# B&R Automation Studio project 305841_E00002_AM_0 (part 16)

#### LocalFunctions.st
```iecst
// Calculate the master and slave angles given cut parameters
FUNCTION_BLOCK fbPopulateCamTable
  // **** Condition inputs
  _numPasses := MAX(1, numPasses); // 1 or greater. Otherwise treat as 1
  _finalDepth := ABS(finalDepth); // must be positive
  _finishPassDepth := MIN(MAX(0.0, finishPassDepth), _finalDepth); // must be >= 0.0, <= final depth.
  _cutInAngle := ABS(cutInAngle); // must be positive
  _overCutAngle := ABS(overCutAngle); // must be positive

  // **** First entry in table is 0,0
  // Axes start at 0,0 (0 offset) at the same velocity (which will normally be zero)
  // Specify absolute positions
  camTable.Section[0].Mode := mcCAMSECTREF_ABSOLUTE;
  camTable.Section[0].MasterPoint := 0.0;
  camTable.Section[0].SlavePoint := 0.0;
  // slave to be at a constant velocity
  camTable.Section[0].FirstDerivative := 1.0; // velocity ratio
  camTable.Section[0].SecondDerivative := 0.0; // accel ratio
  // next point will be offset. Use polynomial for this -- good general case solution
  camTable.Section[0].Type := mcCAMSECTLAW_5TH_ORDER_POLYNOM;
  camTable.Section[0].InflectionPoint := 0.0; // not used for polynomial

  // **** Figure out pass depths and then resulting angles
  // Make cam table entries
  incrCutDepth := (_finalDepth - _finishPassDepth) / _numPasses;

  IF incrCutDepth > 0.0 THEN
    // normal case where finishing pass < final depth
    FOR passCount := 1 TO _numPasses DO
      // depth for this pass
      totalPassDepth := incrCutDepth * passCount;
      // Look up angle for the needed depth
      fbLookupAngle(xVal := totalPassDepth,
                     t1 := ADR(depthToAngle_T1),
                     t2 := ADR(depthToAngle_T2),
                     t3 := ADR(depthToAngle_T3));
      passAngle := fbLookupAngle.yVal;

      // At this point, we have the angle for this pass.
      // This angle is actually the offset angle between the axes.
      // The offset in practice should be negative, meaning the slave lags
      // behind the master by the amount of the offset.
      // Make an entry in the cam table
      // Each pass has an enrty to establish the pass depth,
      // and a second pass to make the cut, which is 1 revolution from the point the
      // depth is established, plus the overcut distance.
      // For a given pass, the first index/position is: ((pass number - 1) * 2) + 1
      // the second index/position is: first index + 1
      // For a given pass, the first master position is: (cutInAngle + pass number) + ((rev + overcut) * (pass number - 1))
      // the second master position is: first position + rev + overcut
      idx := ((passCount - 1) * 2) + 1; // zero based array index position

      // Establish an offset from previous position
      camTable.Section[idx].Mode := mcCAMSECTREF_ABSOLUTE;
      camTable.Section[idx].MasterPoint := (_cutInAngle * passCount) + ((360.0 + _overCutAngle) * (passCount - 1));
      camTable.Section[idx].SlavePoint := camTable.Section[idx].MasterPoint - passAngle;
      // slave to be at a constant velocity
      camTable.Section[idx].FirstDerivative := 1.0; // velocity ratio
      camTable.Section[idx].SecondDerivative := 0.0; // accel ratio
      // next point will be a stright section.
      camTable.Section[idx].Type := mcCAMSECTLAW_STRAIGHT_LINE;
      camTable.Section[idx].InflectionPoint := 0.0; // not used for straight line

      // Keep the offset for a revolution + the overcut distance
      camTable.Section[idx + 1].Mode := mcCAMSECTREF_ABSOLUTE;
      camTable.Section[idx + 1].MasterPoint := camTable.Section[idx].MasterPoint + (360.0 + _overCutAngle);
      camTable.Section[idx + 1].SlavePoint := camTable.Section[idx + 1].MasterPoint - passAngle;
      // slave to be at a constant velocity
      camTable.Section[idx + 1].FirstDerivative := 1.0; // velocity ratio
      camTable.Section[idx + 1].SecondDerivative := 0.0; // accel ratio
      // next point will establish a new offset, so use a polynomial
      camTable.Section[idx + 1].Type := mcCAMSECTLAW_5TH_ORDER_POLYNOM;
      camTable.Section[idx + 1].InflectionPoint := 0.0; // not used for polynomial
    END_FOR;
  ELSE
    // Special case where finishing pass was entered to be >= final depth.
    // Nothing to do, and this else is here for documentation and as
    // a place holder in case something ends up being needed.
    // The finishing pass is handled next, and will cover this case
    ;
  END_IF

  // **** Figure out finishing pass situation

  // If there is a finishing pass, then create cam entries for it

  // After the for loop, passCount will be 1 more than the number of passes.
  // Perfect for the finishing pass, or the retract entry.
  idx := ((passCount - 1) * 2) + 1; // zero based array index position
  IF _finishPassDepth > 0.0 THEN
    // There is a finishing pass
    // By definition, the finishing pass gets us to our final depth,
    // so regardless of the earlier passes, the finishing pass is always
    // at the offset to give the final depth.
    // Look up angle for the needed depth
    fbLookupAngle(xVal := _finalDepth,
                   t1 := ADR(depthToAngle_T1),
                   t2 := ADR(depthToAngle_T2),
                   t3 := ADR(depthToAngle_T3));
    passAngle := fbLookupAngle.yVal;

    // Establish an offset from previous position
    camTable.Section[idx].Mode := mcCAMSECTREF_ABSOLUTE;
    camTable.Section[idx].MasterPoint := (_cutInAngle * passCount) + ((360.0 + _overCutAngle) * (passCount - 1));
    camTable.Section[idx].SlavePoint := camTable.Section[idx].MasterPoint - passAngle;
    // slave to be at a constant velocity
    camTable.Section[idx].FirstDerivative := 1.0; // velocity ratio
    camTable.Section[idx].SecondDerivative := 0.0; // accel ratio
    // next point will be a stright section.
    camTable.Section[idx].Type := mcCAMSECTLAW_STRAIGHT_LINE;
    camTable.Section[idx].InflectionPoint := 0.0; // not used for straight line

    // Keep the offset for a revolution + the overcut distance
    camTable.Section[idx + 1].Mode := mcCAMSECTREF_ABSOLUTE;
    camTable.Section[idx + 1].MasterPoint := camTable.Section[idx].MasterPoint + (360.0 + _overCutAngle);
    camTable.Section[idx + 1].SlavePoint := camTable.Section[idx + 1].MasterPoint - passAngle;
    // slave to be at a constant velocity
    camTable.Section[idx + 1].FirstDerivative := 1.0; // velocity ratio
    camTable.Section[idx + 1].SecondDerivative := 0.0; // accel ratio
    // next point will establish a new offset, so use a polynomial
    camTable.Section[idx + 1].Type := mcCAMSECTLAW_5TH_ORDER_POLYNOM;
    camTable.Section[idx + 1].InflectionPoint := 0.0; // not used for polynomial

    // increment the pass count so similar it can be used for the last entry
    passCount := passCount + 1;
    // calculate a new index for the last entry, which retracts the cutter
    idx := ((passCount - 1) * 2) + 1; // zero based array index position
  END_IF;

  // **** Do the last entry to retract the cutting head.
  // passCount will either be number of passes + 1 in the non-finishing pass case,
  // or will be number of passes + 2 in the finishing pass case. idx and passCount
  // were already adjusted in the finishing pass case.

  // The last cam entry needs to be of type mcCAMSECTLAW_LAST_POINT
  // Establish a zero offset from previous position
  camTable.Section[idx].Mode := mcCAMSECTREF_ABSOLUTE;
  camTable.Section[idx].MasterPoint := (_cutInAngle * passCount) + ((360.0 + _overCutAngle) * (passCount - 1));
  camTable.Section[idx].SlavePoint := camTable.Section[idx].MasterPoint;
  // slave to be at a constant velocity
  camTable.Section[idx].FirstDerivative := 1.0; // velocity ratio
  camTable.Section[idx].SecondDerivative := 0.0; // accel ratio
  // next point will be a stright section.
  camTable.Section[idx].Type := mcCAMSECTLAW_LAST_POINT;
  camTable.Section[idx].InflectionPoint := 0.0; // not used for straight line

END_FUNCTION_BLOCK

FUNCTION_BLOCK fbLookUpYValT3
  // See what table the x value is in
  tableNumber := fctGetTableNumberT3(xVal, ADR(t1), ADR(t2), ADR(t2));
  // Look up the angle (y value) from the correct table
  // The fbDepthToAngle will interpolate between table entries
  IF 1 = tableNumber THEN
    // Set up the lookup fb
    fbDepthToAngleLu(Enable := FALSE);
    fbDepthToAngleLu.NumberOfNodes := t1.numberOfVals;
    fbDepthToAngleLu.NodeVectorX := t1.xVals;
    fbDepthToAngleLu.FcnValues := t1.yVals;
    fbDepthToAngleLu.InX := xVal;
    // look up the Y value
    fbDepthToAngleLu(Enable := TRUE);
    IF fbDepthToAngleLu.Enable AND NOT fbDepthToAngleLu.Error THEN
      // Lookup worked. Send out the looked up value.
      yVal := fbDepthToAngleLu.Out;
    ELSE
      // Lookup didn't work. Send ou the sentinel value.
      yVal := INVALID_SENTINEL;
    END_IF;

  ELSIF 2 = tableNumber THEN
    // Set up the lookup fb
    fbDepthToAngleLu(Enable := FALSE);
    fbDepthToAngleLu.NumberOfNodes := t2.numberOfVals;
    fbDepthToAngleLu.NodeVectorX := t2.xVals;
    fbDepthToAngleLu.FcnValues := t2.yVals;
    fbDepthToAngleLu.InX := xVal;
    // look up the Y value
    fbDepthToAngleLu(Enable := TRUE);
    IF fbDepthToAngleLu.Enable AND NOT fbDepthToAngleLu.Error THEN
      // Lookup worked. Send out the looked up value.
      yVal := fbDepthToAngleLu.Out;
    ELSE
      // Lookup didn't work. Send ou the sentinel value.
      yVal := INVALID_SENTINEL;
    END_IF;

  ELSIF 3 = tableNumber THEN
    // Set up the lookup fb
    fbDepthToAngleLu(Enable := FALSE);
    fbDepthToAngleLu.NumberOfNodes := t3.numberOfVals;
    fbDepthToAngleLu.NodeVectorX := t3.xVals;
    fbDepthToAngleLu.FcnValues := t3.yVals;
    fbDepthToAngleLu.InX := xVal;
    // look up the Y value
    fbDepthToAngleLu(Enable := TRUE);
    IF fbDepthToAngleLu.Enable AND NOT fbDepthToAngleLu.Error THEN
      // Lookup worked. Send out the looked up value.
      yVal := fbDepthToAngleLu.Out;
    ELSE
      // Lookup didn't work. Send ou the sentinel value.
      yVal := INVALID_SENTINEL;
    END_IF;
  END_IF;

END_FUNCTION_BLOCK

// Given an X, find which of 3 tables to look in
FUNCTION fctGetTableNumberT3
  // Return a 1, 2, or 3 for which table to look in
  // NOTE: X values in each table need to be sorted in ascending order
  // NOTE: It is assumed that x values in table 1 < table 2 < table 3

  // If value is less than or equal the last value in table 1,
  // then the value must represented in or before table 1. Return 1.
  IF xVal <= t1.xVals[t1.numberOfVals - 1] THEN
    fctGetTableNumberT3 := 1;
    RETURN;
  ELSIF xVal >= t3.xVals[0] THEN
    // If value is greater than or equal to the first value in table 3,
    // then the value must be represented in or after table 3. Return 3.
    fctGetTableNumberT3 := 3;
    RETURN;
  ELSE
    // The value must be too big to be represented in table 1,
    // and too small to be represented in table 3.
    // Table 2 is the best choice. Return 2.
    fctGetTableNumberT3 := 2;
    RETURN;
  END_IF;

END_FUNCTION

// Given a table, swap the X and Y values
FUNCTION fctSwapTableT3
  // Make sure number of values does not overrun the array sizes
  length := MIN(SIZEOF(tVals) / SIZEOF(tVals[0]), SIZEOF(table.xVals) / SIZEOF(table.xVals[0]), SIZEOF(table.yVals) / SIZEOF(table.yVals[0]));
  // Y -> temp
  // X -> Y
  // temp -> X
  // nextAddr := brsmemcpy(ADR(Dest),ADR(Src),length);
  nextAddr := brsmemcpy(ADR(tVals), ADR(table.yVals), length);
  nextAddr := brsmemcpy(ADR(table.yVals), ADR(table.xVals), length);
  nextAddr := brsmemcpy(ADR(table.xVals), ADR(tVals), length);
END_FUNCTION
```

### Library Logical/PlcLogic/CutProfile/CreateCamTable

#### CreateCamTable.var
```iecst
VAR CONSTANT
  CAM_POINTS : UINT := 250;
END_VAR

VAR

  (* program control *)
  seqCtr : SINT; (* sequence counter *)
  idx : UINT; (* index *)

  (****** Cam related ******)
  (* program control for cam creation *)
  reqCreateCamTable : BOOL := FALSE; (* request to start seq *)
  createCamTableOS : BOOL := FALSE;
  createCamTableDone : BOOL := FALSE;
  camTableId : UINT := 14; (* 1-14, but data type compatible with cam prepare fb *)
  camSeqCtr : SINT; (* sequence counter *)
  camTable : McCamSectionsType; (* local cam sections table *)
  camData : McCamDataType; (* cam data calculated from sections *)
  camPointsMaster : ARRAY[0..CAM_POINTS] OF LREAL;
  camPointsSlave : ARRAY[0..CAM_POINTS] OF LREAL;
  fbCreateCamSections : fbCalcCamSections;
  fbCalcCamFromSections : MC_BR_CalcCamFromSections;
  fbCalcCamPoints : MC_BR_CalcPointsFromCam;
  fbCamPrepare : MC_BR_CamPrepare;
  (* detect changes to cut profile *)
  cutProfilePrev : sWp_CuttingHead;
  (* BR Str mem fct params *)
  cutProfileBytes : UDINT;
  result : DINT;
  nxtAddr : UDINT;

  (****** Recipe and file related ******)

  (* Local version OF the lookup table *)
	depthToAngleLu : sDepthToAngleLu;

  (* program control for directory creation *)
  reqInitDirs : BOOL := FALSE; (* request to start seq *)
  initDirsOS : BOOL := FALSE;
  initDirsDone : BOOL := FALSE;
  devName : STRING[80]; (* also used for recipe read *)
  dirName : STRING[255];

  (* program control for Depth To Angle Lu recipe registration *)
  pvNameLocalDepthToAngleLu : STRING[100];
  pvNameGloballDepthToAngleLu : STRING[100];
  pvCatagoryDepthToAngleLu : STRING[50];

  (* program control for recipe read/write *)
  recipeReadOverwiteGlobal : BOOL := FALSE;

  recipeReadFileName : STRING[255];
  recipeWriteFileName : STRING[255];

  reqRecipeReadAngleLu : BOOL := FALSE;
  recipeReadAngleLuOS : BOOL := FALSE;
  recipeReadAngleLuDone : BOOL := FALSE;

  reqRecipeWriteAngleLu : BOOL := FALSE;
  recipeWriteAngleLuOS : BOOL := FALSE;
  recipeWriteAngleLuDone : BOOL := FALSE;
  csvHeader : MpRecipeCsvHeaderType;

  (* FileIO fbs *)
  fbDirCreate : DirCreate;

  (* recipe fbs *)
  fbRcpiRegLocalDToALu : MpRecipeRegPar; (* register local Depth To Angle Lu Table to recipe *)
  fbRcpiRegGlobalDToALu : MpRecipeRegPar; (* register global Depth To Angle Lu Table to recipe *)
  fbRecipeCsv : MpRecipeCsv; (* recipe to/from file *)

END_VAR
```

#### LocalFunctions.fun
```iecst
FUNCTION_BLOCK fbLookUpYValT3 (* Given an X, get the possibly interpolated value for Y *)
	VAR CONSTANT
		INVALID_SENTINEL : REAL := -9999.0;
	END_VAR

	VAR_INPUT
    LoadTables : BOOL; (* load lookup table values *)
    Enable : BOOL; (* trigger a lookup *)
		XVal : REAL; (* x value to lookup *)
		T1 : REFERENCE TO sXYTableReal50; (* table 1 *)
		T2 : REFERENCE TO sXYTableReal50; (* table 2 *)
		T3 : REFERENCE TO sXYTableReal50; (* table 3 *)
	END_VAR

	VAR_OUTPUT
    IsTablesLoaded : BOOL; (* look up tables have been loaded *)
    Active : BOOL;
    Done : BOOL;
    Error : BOOL;
		YVal : REAL; (* looked up and interpolated Y value *)
	END_VAR

	VAR
    (* oneshots *)
    _loadOS : BOOL := FALSE;
    _enableOS : BOOL := FALSE;
    (* which table to use *)
		_xValPrev : REAL; (* previous x value to lookup *)
    _tableNumber : USINT;
    (* table lookup fbs*)
		_fbDepthToAngleLuT1 : MTLookUpTable;
		_fbDepthToAngleLuT2 : MTLookUpTable;
		_fbDepthToAngleLuT3 : MTLookUpTable;
	END_VAR
END_FUNCTION_BLOCK

FUNCTION_BLOCK fbPopulateCamSections (* Calculate the master and slave angles given cut parameters *)
	VAR_INPUT
    Enable : BOOL;
		PassCount : USINT := 1; (* number of passes *)
		FinalDepth : REAL; (* final cut depth, in units of lookup table *)
		FinishPassDepth : REAL := 0.0; (* finishing pass depth. In units of lookup table. Set to 0 for no finish pass. *)
		CutInAngle : REAL; (* degrees *)
		OverCutAngle : REAL; (* degrees *)
		CamTable : REFERENCE TO McCamSectionsType; (* X values master angle, Y values slave angle *)
		DepthToAngle_T1 : REFERENCE TO sXYTableReal50;
		DepthToAngle_T2 : REFERENCE TO sXYTableReal50;
		DepthToAngle_T3 : REFERENCE TO sXYTableReal50;
	END_VAR

  VAR_OUTPUT
    Active : BOOL := FALSE;
    Done : BOOL := FALSE;
    Error : BOOL := FALSE;
  END_VAR

	VAR
    enableOS : BOOL := FALSE;
		_numPasses : USINT; (* conditioned number of passes *)
		_finalDepth : REAL; (* conditioned final cut depth *)
		_finishPassDepth : REAL; (* conditioned finishing pass depth. Set to 0 for no finish pass. *)
		_cutInAngle : REAL; (* conditioned value *)
		_overCutAngle : REAL; (* conditioned value *)
    seqCtr : SINT; (* sequence counter *)
		passCtr : USINT; (* pass counter *)
		incrCutDepth : REAL; (* incremental depth of a nominal pass *)
		totalPassDepth : REAL; (* accum depth for the pass *)
		passAngle : REAL;
		idx : USINT; (* index *)
    (* lookup angle from depth fb *)
    fbLookupAngle : fbLookUpYValT3;
	END_VAR
END_FUNCTION_BLOCK

FUNCTION fctGetTableNumberT3 : USINT (* Given an X, find which table to look in *)
	VAR_INPUT
		xVal : REAL;
		t1 : REFERENCE TO sXYTableReal50; (* table 1 *)
		t2 : REFERENCE TO sXYTableReal50; (* table 2 *)
		t3 : REFERENCE TO sXYTableReal50; (* table 3 *)
	END_VAR
END_FUNCTION

FUNCTION fctSwapTableT3 : USINT (* Swap X & Y columns *)
	VAR_INPUT
		table : REFERENCE TO sXYTableReal50; (* table to swap the X & Y values of *)
	END_VAR
	VAR
		tVals : ARRAY[0..49] OF REAL; (* temporary storage *)
		length : UDINT; (* mem copy length in bytes *)
		nextAddr : UDINT; (* return from memcpy *)
	END_VAR
END_FUNCTION
```

#### CreateCamTable.st
```iecst
PROGRAM _INIT

  (****** Cam related ******)
  // Set up fb to populate cam sections
  fbCreateCamSections.CamTable := ADR(camTable);
  fbCreateCamSections.DepthToAngle_T1 := ADR(gr_depthToAngleLu.T1);
  fbCreateCamSections.DepthToAngle_T2 := ADR(gr_depthToAngleLu.T2);
  fbCreateCamSections.DepthToAngle_T3 := ADR(gr_depthToAngleLu.T3);

  (****** Recipe and file related ******)
  gr_depthToAngleLu; // Make sure the tables exist!!
  depthToAngleLu;

  // Setup registration of PV to a recipe
  // Each PV uses a separate registration FB
  // Local Depth To Angle LU Table
  // Use local LU table for recipe access and transfer to/from global when all is well
  pvNameLocalDepthToAngleLu := 'CrCamTbl:depthToAngleLu';
  pvCatagoryDepthToAngleLu := 'DepthToAngle';
  fbRcpiRegLocalDToALu.MpLink := ADR(angleLuRecipeCsv);
  fbRcpiRegLocalDToALu.Enable := FALSE;
  fbRcpiRegLocalDToALu.ErrorReset := FALSE;
  fbRcpiRegLocalDToALu.PVName := ADR(pvNameLocalDepthToAngleLu);
  fbRcpiRegLocalDToALu.Category := ADR(pvCatagoryDepthToAngleLu);
  // set up the fb by calling with enable false, and then set enable
  // true so it is ready to go in cyclic.
  fbRcpiRegLocalDToALu();
  fbRcpiRegLocalDToALu.Enable := TRUE;

  // Global Depth To Angle LU Table
  // Use local LU table for recipe access and transfer to/from global when all is well
  pvNameGloballDepthToAngleLu := 'gr_depthToAngleLu';
  pvCatagoryDepthToAngleLu := 'DepthToAngle';
  fbRcpiRegGlobalDToALu.MpLink := ADR(angleLuRecipeCsv);
  fbRcpiRegGlobalDToALu.Enable := FALSE;
  fbRcpiRegGlobalDToALu.ErrorReset := FALSE;
  fbRcpiRegGlobalDToALu.PVName := ADR(pvNameGloballDepthToAngleLu);
  fbRcpiRegGlobalDToALu.Category := ADR(pvCatagoryDepthToAngleLu);
  // set up the fb by calling with enable false, and then set enable
  // true so it is ready to go in cyclic.
  fbRcpiRegGlobalDToALu();
  fbRcpiRegGlobalDToALu.Enable := TRUE;

  // Set flag to create directories
  initDirs := TRUE; // true will trigger dir setup (creation) after startup
  initDirsOS := FALSE;
  initDirsDone := FALSE;

  // Set flags to control read/write of recipes
  // recipe file names
  recipeReadFileName := 'DepthToAngleLookup_recipe_b.csv';
  recipeWriteFileName := 'DepthToAngleLookup_recipe_b_FromPlc.csv';

  // set whether or not to overwrite the global data on sucessful local read
  recipeReadOverwiteGlobal := FALSE;

  recipeReadAngleLu := FALSE; // set high to read recipe after startup
  recipeReadAngleLuOS := FALSE;
  recipeReadAngleLuDone := FALSE;

  recipeWriteAngleLu := FALSE; // set high to read recipe after startup
  recipeWriteAngleLuOS := FALSE;
  recipeWriteAngleLuDone := FALSE;

 END_PROGRAM

PROGRAM _CYCLIC

  // *****************
  // Create Cam table on request
  // *****************

  // On request, calculate and populate cam sections base on cut parameters.
  // Done sucessfully, and camSeqCtr should start from 1, go up, and then end up at -1.
  // Errors result in a more negative camSeqCtr
  // TODO: Deal with errors. Right now the sequence stops, with the camSeqCtr being set to
  // a value more negative than -1.

  IF createCamTable THEN

    // if the OS is clear, this is the first time thru ...
    // init the seq number and manage flags and OS
    IF NOT createCamTableOS THEN
      // Set the OS so this bit only happens once per req
      createCamTableOS := TRUE;
      // Init the seq ctr
      camSeqCtr := 1;
      // Clear the done flag
      createCamTableDone := FALSE;
    END_IF;

    IF 1 = camSeqCtr THEN
      // Use cam id 14 for calculated cam table
      camTableId := 14;

      // Set up to calc the cam sections fb
      // Use the current cutting head configuration for the cut profile

      // Force the finish pass depth to be zero if the option is not chosen
      IF gr_CfgCurrent.cuttingHead.finishingPass THEN
        fbCreateCamSections.FinishPassDepth :=  gr_CfgCurrent.cuttingHead.finishingPassDepth;
      ELSE
        fbCreateCamSections.FinishPassDepth := 0.0;
      END_IF;
      fbCreateCamSections.PassCount := gr_CfgCurrent.cuttingHead.passCount;
      fbCreateCamSections.FinalDepth := gr_CfgCurrent.cuttingHead.totalDepth;
      fbCreateCamSections.CutInAngle :=  LREAL_TO_REAL(gr_CfgCurrent.cuttingHead.depthAdjAngle);
      fbCreateCamSections.OverCutAngle :=  LREAL_TO_REAL(gr_CfgCurrent.cuttingHead.cutOverrunAngle);

      // Clear the camTable, camData, and point arrays
      // nxt_adr := brsmemset(ADR(Mem),value,length);
      nxtAddr := brsmemset(ADR(camTable), 0, SIZEOF(camTable));
      nxtAddr := brsmemset(ADR(camData), 0, SIZEOF(camData));
      nxtAddr := brsmemset(ADR(camPointsMaster), 0, SIZEOF(camPointsMaster));
      nxtAddr := brsmemset(ADR(camPointsSlave), 0, SIZEOF(camPointsSlave));

      // Call with enable false to make sure everything is reset and ready to execute with new info
      fbCreateCamSections.Enable := FALSE;
      fbCreateCamSections();
      // onto the next step
      camSeqCtr := 2;
    ELSIF 2 = camSeqCtr THEN
      // Calc the cam sections
      fbCreateCamSections.Enable := TRUE;
      fbCreateCamSections();
      IF fbCreateCamSections.Done AND NOT fbCreateCamSections.Error THEN
        // All done and no error. Move on ...
        // Reset FB and go to next step
        fbCreateCamSections.Enable := FALSE;
        fbCreateCamSections();
        camSeqCtr := 3;
      ELSIF fbCreateCamSections.Done AND fbCreateCamSections.Error THEN
        // Done with an error. Bail out ...
        camSeqCtr := -2;
      END_IF;
    ELSIF 3 = camSeqCtr THEN
      // Set up to calc the cam from the sections
      fbCalcCamFromSections.CamSectionsAddress := ADR(camTable);
      fbCalcCamFromSections.CamDataAddress := ADR(camData);
      // Call with execute false to make sure everything is reset and ready to execute with new info
      fbCalcCamFromSections.Execute := FALSE;
      fbCalcCamFromSections();
      // onto the next step
      camSeqCtr := 4;
    ELSIF 4 = camSeqCtr THEN
      // Calc the cam sections
      fbCalcCamFromSections.Execute := TRUE;
      fbCalcCamFromSections();
      IF fbCalcCamFromSections.Done AND NOT fbCalcCamFromSections.Error THEN
        // All done and no error. Move on ...
        // Reset FB and go to next step
        fbCalcCamFromSections.Execute := FALSE;
        fbCalcCamFromSections();
        camSeqCtr := 5;
      ELSIF NOT fbCalcCamFromSections.Busy AND fbCalcCamFromSections.Error THEN
        // Done with an error. Bail out ...
        camSeqCtr := -4;
      END_IF;
    ELSIF 5 = camSeqCtr THEN
      // Set up to prepare and load the cam data
      fbCamPrepare.Axis := ADR(axes[AD_INNER_ECCENTRIC].AxisObj);
      fbCamPrepare.Cam.DataObjectName := ''; // not used if Cam.DataAdress <> 0
      fbCamPrepare.Cam.DataAdress := ADR(camData); // cam data calculated in fbCalcCamFromSections
      fbCamPrepare.CamID := camTableId;
      // Call with execute false to make sure everything is reset and ready to execute with new info
      fbCamPrepare.Execute := FALSE;
      fbCamPrepare();
      // onto the next step
      camSeqCtr := 6;
    ELSIF 6 = camSeqCtr THEN
      // Prepare and load the cam data
      fbCamPrepare.Execute := TRUE;
      fbCamPrepare();
      IF fbCamPrepare.Done AND NOT fbCamPrepare.Error THEN
        // All done and no error. Move on ...
        // Reset FB and go to next step
        fbCamPrepare.Execute := FALSE;
        fbCamPrepare();
        camSeqCtr := -1;  // TEST: skip fbCalcCamPoints. Getting an error
      ELSIF NOT fbCamPrepare.Busy AND fbCamPrepare.Error THEN
        // Done with an error. Bail out ...
        camSeqCtr := -6;
      END_IF;
    ELSIF 7 = camSeqCtr THEN
      // Set up to calculate cam points
      fbCalcCamPoints.Cam.DataObjectName := ''; // not used if Cam.DataAdress <> 0
      fbCalcCamPoints.Cam.DataAdress := ADR(camData); // cam data calculated in fbCalcCamFromSections
      fbCalcCamPoints.MasterPointsAddress := ADR(camPointsMaster);
      fbCalcCamPoints.SlavePointsAddress := ADR(camPointsSlave);
      fbCalcCamPoints.NumberOfPoints := CAM_POINTS;
      // Call with execute false to make sure everything is reset and ready to execute with new info
      fbCalcCamPoints.Execute := FALSE;
      fbCalcCamPoints();
      // onto the next step
      camSeqCtr := 8;
    ELSIF 8 = camSeqCtr THEN
      // Calcuate points from the cam data
      fbCalcCamPoints.Execute := TRUE;
      fbCalcCamPoints();
      IF fbCalcCamPoints.Done AND NOT fbCalcCamPoints.Error THEN
        // All done and no error. Move on ...
        // reset fb
        fbCalcCamPoints.Execute := FALSE;
        fbCalcCamPoints();
        camSeqCtr := -1;
      ELSIF NOT fbCalcCamPoints.Busy AND fbCalcCamPoints.Error THEN
        // Done with an error. Bail out ...
        camSeqCtr := -8;
      END_IF;
    ELSIF -1 = camSeqCtr THEN
      // All done making cam sections.
      // Getting ready if another request is made.
      // Clear the createCamTable flag and OS and set the done.
     createCamTable := FALSE;
     createCamTableOS := FALSE; // clear the OS so another initDirs resets things up top
     createCamTableDone := TRUE;
     // reset fb
     fbCreateCamSections.Enable := FALSE;
     fbCreateCamSections();
    END_IF;
  ELSE
    // createCamTable is false. Clear the OS so we can one time thru it next time
    createCamTableOS := FALSE;
  END_IF;

  // *****************
  // Set up directories
  // *****************
  // Execute FileIO DirCreate async until done or error
  // seqCtr odd: set up DirCreate fb
  // seqCtr even : create dir
  // Use the OS so the directory management can be easily re-run
  // by setting initDirs true (again)
  IF initDirs THEN
    // if the OS is clear, this is the first time thru ...
    // init the seq number and manage flags and OS
    IF NOT initDirsOS THEN
      // Set the OS so this bit only happens once per initDirs
      initDirsOS := TRUE;
      // Init the seq ctr
      seqCtr := 1;
      // Clear the done flag
      initDirsDone := FALSE;
    END_IF;

    IF 1 = seqCtr THEN
      // Setup for first dir
      devName := 'UserPartitionRoot';
      dirName := 'config';
      fbDirCreate.enable := FALSE;
      fbDirCreate.pDevice := ADR(devName);
      fbDirCreate.pName := ADR(dirName);
      fbDirCreate();
      IF ERR_FUB_ENABLE_FALSE = fbDirCreate.status THEN
        seqCtr := 2;
      END_IF;
    ELSIF 2 = seqCtr THEN
      // create first dir
      fbDirCreate.enable := TRUE;
      fbDirCreate();
      IF ERR_OK = fbDirCreate.status OR fiERR_DIR_ALREADY_EXIST = fbDirCreate.status THEN
        // creation okay or not needed
        seqCtr := 3;
      END_IF;
    ELSIF 3 = seqCtr THEN
      // Setup for seconnd dir
      dirName := 'config\recipes';
      // same addresses for device and name
      fbDirCreate.enable := FALSE;
      fbDirCreate();
      IF ERR_FUB_ENABLE_FALSE = fbDirCreate.status THEN
        seqCtr := 4;
      END_IF;
    ELSIF 4 = seqCtr THEN
      // create second dir
      fbDirCreate.enable := TRUE;
      fbDirCreate();
      IF ERR_OK = fbDirCreate.status OR fiERR_DIR_ALREADY_EXIST = fbDirCreate.status THEN
        // creation okay or not needed
        seqCtr := -1;
      END_IF;
    ELSIF -1 = seqCtr THEN
      // All done making directories.
      // Getting ready if another request is made.
      // Clear the initDirs flag and OS and set the done.
     initDirs := FALSE;
     initDirsOS := FALSE; // clear the OS so another initDirs resets things up top
     initDirsDone := TRUE;
     // shut off the fb as a matter of good practice
     fbDirCreate.enable := FALSE;
     fbDirCreate();
    END_IF;
  ELSE
    // initDirs is false. Clear the OS so we can one time thru it next time
    initDirsOS := FALSE;
  END_IF;

  // *****************
  // Read Write Lu Tables to/from recipe
  // *****************

  // Recipe Registration fb should be called all the time, and need to be active
  // when recipe read/write is performed.
  // MpRecipeRegPar was set up in init
  fbRcpiRegLocalDToALu();
  fbRcpiRegGlobalDToALu();

  // **** Read Recipe
  // Treat recipe read as async until done or error
  // seqCtr odd: set up fbRecipeCsv fb
  // seqCtr even : read recipe
  // Use the OS so the read can be easily re-run
  // by setting registerPvs true (again)
  IF NOT initDirs AND initDirsDone AND
      fbRcpiRegLocalDToALu.Active AND NOT fbRcpiRegLocalDToALu.Error AND
      fbRcpiRegGlobalDToALu.Active AND NOT fbRcpiRegGlobalDToALu.Error AND
      recipeReadAngleLu AND NOT recipeWriteAngleLu THEN
    // if the OS is clear, this is the first time thru ...
    // init the seq number and manage flags and OS
    IF NOT recipeReadAngleLuOS THEN
      // Set the OS so this bit only happens once per initDirs
      recipeReadAngleLuOS := TRUE;
      // Set the pv number
      seqCtr := 1;
      // Clear the done flag
      recipeReadAngleLuDone := FALSE;
    END_IF;

    IF 1 = seqCtr THEN
      // Setup for first pv
      devName := 'Recipes';
      pvCatagoryDepthToAngleLu := 'DepthToAngle';
      fbRecipeCsv.MpLink := ADR(angleLuRecipeCsv);
      fbRecipeCsv.Enable := FALSE;
      fbRecipeCsv.ErrorReset := FALSE;
      fbRecipeCsv.DeviceName := ADR(devName);
      fbRecipeCsv.FileName := ADR(recipeReadFileName);
      fbRecipeCsv.Header := ADR(csvHeader);
      fbRecipeCsv.Category := ADR(pvCatagoryDepthToAngleLu);
      fbRecipeCsv.LoadType := mpRECIPE_CSV_LOAD_ALL;
      fbRecipeCsv.Load := TRUE;
      fbRecipeCsv.Save := FALSE;
      fbRecipeCsv.UpdateNotification := FALSE;
      fbRecipeCsv();
      IF NOT fbRecipeCsv.Enable AND NOT fbRecipeCsv.Active AND 0 = fbRecipeCsv.StatusID THEN
        seqCtr := 2;
      END_IF;
    ELSIF 2 = seqCtr THEN
      // read the recipe file and populate the pv
      fbRecipeCsv.Enable := TRUE;
      fbRecipeCsv();
      IF fbRecipeCsv.CommandDone AND NOT fbRecipeCsv.Error THEN
        // read ok
        // If the bit is set, transfer local to the global table -- thisglobal is battery backed retained/permanent
        IF recipeReadOverwiteGlobal THEN
          gr_depthToAngleLu := depthToAngleLu;
        END_IF;
        seqCtr := -1; // all done!
      END_IF;
    ELSIF -1 = seqCtr THEN
      // All done reading the recipe. Deal with flags
      recipeReadAngleLu := FALSE;
      recipeReadAngleLuOS := FALSE; // clear the OS so another registerPv resets things
      recipeReadAngleLuDone := TRUE;
      // shut off the fb as a matter of good practice
      fbRecipeCsv.Enable := FALSE;
      fbRecipeCsv();
    END_IF;
  ELSE
    // Earlier operations not done, or recipeReadAngleLu flag is clear. Clear to OS so we can one time thru it next time
    recipeReadAngleLuOS := FALSE;
  END_IF;

  // **** Write Recipe
  // Treat recipe read as async until done or error
  // seqCtr odd: set up fbRecipeCsv fb
  // seqCtr even : read recipe
  // Use the OS so the read can be easily re-run
  // by setting registerPvs true (again)
  IF NOT initDirs AND initDirsDone AND
      fbRcpiRegLocalDToALu.Active AND NOT fbRcpiRegLocalDToALu.Error AND
      fbRcpiRegGlobalDToALu.Active AND NOT fbRcpiRegGlobalDToALu.Error AND
      recipeWriteAngleLu AND NOT recipeReadAngleLu THEN
    // if the OS is clear, this is the first time thru ...
    // init the seq number and manage flags and OS
    IF NOT recipeWriteAngleLuOS THEN
      // Set the OS so this bit only happens once per initDirs
      recipeWriteAngleLuOS := TRUE;
      // Set the pv number
      seqCtr := 1;
      // Clear the done flag
      recipeWriteAngleLuDone := FALSE;
    END_IF;

    IF 1 = seqCtr THEN
      // Setup for first pv
      devName := 'Recipes';
      pvCatagoryDepthToAngleLu := 'DepthToAngle';
      csvHeader.Name := 'DepthToAngle';
      csvHeader.Description := 'Depths are given in inches, and angles correspond to negative (slave lag) offsets. Source is Robbie Potts Email.';
      csvHeader.Version := 'b';
      csvHeader.DateTime := DT#2022-06-03-14:56;
      fbRecipeCsv.MpLink := ADR(angleLuRecipeCsv);
      fbRecipeCsv.Enable := FALSE;
      fbRecipeCsv.ErrorReset := FALSE;
      fbRecipeCsv.DeviceName := ADR(devName);
      fbRecipeCsv.FileName := ADR(recipeWriteFileName);
      fbRecipeCsv.Header := ADR(csvHeader);
      fbRecipeCsv.Category := ADR(pvCatagoryDepthToAngleLu);
      fbRecipeCsv.LoadType := mpRECIPE_CSV_LOAD_ALL;
      fbRecipeCsv.Load := FALSE;
      fbRecipeCsv.Save := TRUE;
      fbRecipeCsv.UpdateNotification := FALSE;
      fbRecipeCsv();
      IF NOT fbRecipeCsv.Enable AND NOT fbRecipeCsv.Active AND 0 = fbRecipeCsv.StatusID THEN
        seqCtr := 2;
      END_IF;
    ELSIF 2 = seqCtr THEN
      // write pv to recipe file
      fbRecipeCsv.Enable := TRUE;
      fbRecipeCsv();
      IF fbRecipeCsv.CommandDone AND NOT fbRecipeCsv.Error THEN
        // read ok
        seqCtr := -1; // all done!
      END_IF;
    ELSIF -1 = seqCtr THEN
      // All done reading the recipe. Deal with flags
      recipeWriteAngleLu := FALSE;
      recipeWriteAngleLuOS := FALSE; // clear the OS so another registerPv resets things
      recipeWriteAngleLuDone := TRUE;
      // shut off the fb as a matter of good practice
      fbRecipeCsv.Enable := FALSE;
      fbRecipeCsv();
    END_IF;
  ELSE
    // Earlier operations not done, or recipeWriteAngleLu flag is clear. Clear to OS so we can one time thru it next time
    recipeWriteAngleLuOS := FALSE;
  END_IF;

END_PROGRAM

PROGRAM _EXIT
	(* Insert code here *)

END_PROGRAM
```

#### LocalFunctions.st
```iecst
FUNCTION_BLOCK fbLookUpYValT3
  // The lookup table needs to be loaded into the MTLookUpTable fb.
  // We don't want to do this every scan, so use the initTables to
  // trigger this, and the isInitialized output to monitor it.
  // Initialize the tables on a rising edge of initTables input,
  // OR if they have not been done yet and the enable goes high.

  IF (LoadTables AND NOT _loadOS) OR (Enable AND NOT IsTablesLoaded) THEN
    // Load tables if requested or if a lookup is triggered and they are not loaded.
    // First set the OS so only a rising edge of loadTables is used
    _loadOS := TRUE;
    // Now load the table values
    _fbDepthToAngleLuT1.NumberOfNodes := T1.numberOfVals;
    _fbDepthToAngleLuT1.NodeVectorX := T1.xVals;
    _fbDepthToAngleLuT1.FcnValues := T1.yVals;

    _fbDepthToAngleLuT2.NumberOfNodes := T2.numberOfVals;
    _fbDepthToAngleLuT2.NodeVectorX := T2.xVals;
    _fbDepthToAngleLuT2.FcnValues := T2.yVals;

    _fbDepthToAngleLuT3.NumberOfNodes := T3.numberOfVals;
    _fbDepthToAngleLuT3.NodeVectorX := T3.xVals;
    _fbDepthToAngleLuT3.FcnValues := T3.yVals;

    // set the output status
    IsTablesLoaded := TRUE;
  ELSIF NOT LoadTables THEN
    // keep OS false when init is not set
    _loadOS := FALSE;
  END_IF;

  // clear the done bit on rising edge of enable
  IF (Enable AND NOT _enableOS) OR (Enable AND XVal <> _xValPrev) THEN
    // first time thru with enable set, or enable is set and the x value changes

    // set the OS
    _enableOS := TRUE;

    // Clear the done bit and set the active bit
    Done := FALSE;
    Active := TRUE;

    // See what table the x value is in
    _tableNumber := fctGetTableNumberT3(XVal, ADR(T1), ADR(T2), ADR(T3));

    // Look up the Y value from the correct table
    // The fbDepthToAngle will interpolate between table entries
    // Call with correct lookup fb with enable false to make sure
    // input changes, including possible table updates above
    // are processed on rising edge of enable later on.
    IF 1 = _tableNumber THEN
      // Set up the lookup fb
      _fbDepthToAngleLuT1.InX := XVal;
      _fbDepthToAngleLuT1.Mode := mtLOOKUP_LINEAR_EXTRAPOLATION;
      _fbDepthToAngleLuT1(Enable := FALSE);
    ELSIF 2 = _tableNumber THEN
      // Set up the lookup fb
      _fbDepthToAngleLuT2.InX := XVal;
      _fbDepthToAngleLuT2.Mode := mtLOOKUP_LINEAR_EXTRAPOLATION;
      _fbDepthToAngleLuT2(Enable := FALSE);
    ELSIF 3 = _tableNumber THEN
      // Set up the lookup fb
      _fbDepthToAngleLuT3.InX := XVal;
      _fbDepthToAngleLuT3.Mode := mtLOOKUP_LINEAR_EXTRAPOLATION;
      _fbDepthToAngleLuT3(Enable := FALSE);
    END_IF;

    // Update the previos X value
    _xValPrev := XVal;

  ELSIF Enable AND _enableOS THEN
    // First time thru completed. Do this while enable is high.
    // LU FBs were set up on first scan thru, so now get on with
    // the lookup.
    IF 1 = _tableNumber THEN
      // look up the Y value from table 1
      _fbDepthToAngleLuT1(Enable := TRUE);
      IF _fbDepthToAngleLuT1.Enable AND _fbDepthToAngleLuT1.Active AND NOT _fbDepthToAngleLuT1.Error THEN
        // Lookup worked. Send out the looked up value.
        YVal := _fbDepthToAngleLuT1.Out;
        Error := FALSE;
      ELSIF _fbDepthToAngleLuT1.Enable AND _fbDepthToAngleLuT1.Error THEN
        // Lookup didn't work. Send out the sentinel value.
        YVal := INVALID_SENTINEL;
        Error := TRUE;
      END_IF;
      // All done, set the done output
      Done := TRUE;
    ELSIF 2 = _tableNumber THEN
      // look up the Y value from table 2
      _fbDepthToAngleLuT2(Enable := TRUE);
      IF _fbDepthToAngleLuT2.Enable AND _fbDepthToAngleLuT2.Active AND NOT _fbDepthToAngleLuT2.Error THEN
        // Lookup worked. Send out the looked up value.
        YVal := _fbDepthToAngleLuT2.Out;
        Error := FALSE;
      ELSIF _fbDepthToAngleLuT2.Enable AND _fbDepthToAngleLuT2.Error THEN
        // Lookup didn't work. Send out the sentinel value.
        YVal := INVALID_SENTINEL;
        Error := TRUE;
      END_IF;
      // All done, set the done output
      Done := TRUE;
    ELSIF 3 = _tableNumber THEN
      // look up the Y value from table 3
      _fbDepthToAngleLuT3(Enable := TRUE);
      IF _fbDepthToAngleLuT3.Enable AND _fbDepthToAngleLuT3.Active AND NOT _fbDepthToAngleLuT3.Error THEN
        // Lookup worked. Send out the looked up value.
        YVal := _fbDepthToAngleLuT3.Out;
        Error := FALSE;
      ELSIF _fbDepthToAngleLuT3.Enable AND _fbDepthToAngleLuT3.Error THEN
        // Lookup didn't work. Send out the sentinel value.
        YVal := INVALID_SENTINEL;
        Error := TRUE;
      END_IF;
      // All done, set the done output
      Done := TRUE;
    ELSE
      // some sort of problem with the table number
      Error := TRUE;
      Done := TRUE;
    END_IF;
  ELSIF NOT Enable THEN
    // Enable is not high. Clear the OS and manage the output stauts
    _enableOS := FALSE;
    Active := FALSE;
    Done := FALSE;
    Error := FALSE;
    // status := ??; TODO: What should status be?
  END_IF;

END_FUNCTION_BLOCK

// Calculate the master and slave angles given cut parameters
FUNCTION_BLOCK fbCalcCamSections
  IF Enable AND NOT enableOS THEN
    // Rising edge of enable ... first time thru.

    // set OS
    enableOS := TRUE;

    // Set active and clear done and error
    Active := TRUE;
    Error := FALSE;
    Done := FALSE;

    // Make sure the lookup tables get loaded in the lookup fb
    // The lookups will come later
    fbLookupAngle.Enable := FALSE;
    fbLookupAngle.T1 := ADR(DepthToAngle_T1);
    fbLookupAngle.T2 := ADR(DepthToAngle_T2);
    fbLookupAngle.T3 := ADR(DepthToAngle_T3);
    fbLookupAngle.LoadTables := TRUE;
    fbLookupAngle();
    fbLookupAngle.LoadTables := FALSE;

    // **** Condition inputs
    _numPasses := MAX(1, PassCount); // 1 or greater. Otherwise treat as 1
    _finalDepth := ABS(FinalDepth); // must be positive
    _finishPassDepth := MIN(MAX(0.0, FinishPassDepth), _finalDepth); // must be >= 0.0, <= final depth.
    _cutInAngle := ABS(CutInAngle); // must be positive
    _overCutAngle := ABS(OverCutAngle); // must be positive

    // Init the seq counter
    seqCtr := 1;

  ELSIF Enable AND enableOS THEN
    // Enable high. Do this stuff over many scans

    IF 1 = seqCtr THEN
      // **** First step: make the first entry and figure out the incremental cut depth

      // **** First entry in table is 0,0
      // At the beginning of the table, it is assumed the axes are at zero offset (0,0)
      // at the same velocity (which will normally be zero)
      // Specify absolute positions
      CamTable.Section[0].Mode := mcCAMSECTREF_ABSOLUTE;
      CamTable.Section[0].MasterPoint := 0.0;
      CamTable.Section[0].SlavePoint := 0.0;
      // slave to be at a constant velocity
      CamTable.Section[0].FirstDerivative := 1.0; // velocity ratio
      CamTable.Section[0].SecondDerivative := 0.0; // accel ratio
      // next point will be offset. Use polynomial for this -- good general case solution
      CamTable.Section[0].Type := mcCAMSECTLAW_5TH_ORDER_POLYNOM;
      CamTable.Section[0].InflectionPoint := 0.0; // not used for polynomial

      // **** Figure out pass depths and then resulting angles
      // Make cam table entries
      incrCutDepth := (_finalDepth - _finishPassDepth) / _numPasses;

      // Ready for the next step
      passCtr := 1; // Init pass counter. If controlled loop in seq step 2/3.
      seqCtr := 2;

    ELSIF 2 = seqCtr OR 3 = seqCtr THEN
      // **** Second step: Lookup the nominal pass angle
      // **** Third step: Calculate the nominal pass angle

      IF incrCutDepth > 0.0 THEN
        // normal case where finishing pass < final depth
        // This would be a FOR loop, but I don't want multi-scan async operations
        // to block or cause scan time issues.
        IF passCtr <= _numPasses THEN
          // depth for this pass
          totalPassDepth := incrCutDepth * passCtr;

          // lookup step
          IF 2 = seqCtr THEN
            // Look up angle for the needed depth
            fbLookupAngle(Enable := TRUE, XVal := totalPassDepth);
            IF fbLookupAngle.Done AND NOT fbLookupAngle.Error THEN
              // Lookup was sucessful. Use the looked up value.
              // Force the angle to be positive, as down below the
              // value is subtracted from the master position to force
              // the slave to have a negative offset.
              // Round just for safety so crazy decimal imprecision or rounding does not cause
              // unexpected small differences in cam entries
              passAngle := fctRound3(_I_src := ABS(fbLookupAngle.YVal));
              // done with LU fb
              fbLookupAngle(Enable := FALSE);
              // move to next step
              seqCtr := 3;
            ELSIF fbLookupAngle.Done AND fbLookupAngle.Error THEN
              // Lookup error. Use 0 for the pass angle, and set the error output
              passAngle := 0.0;
              Error := TRUE;
              // done with LU fb
              fbLookupAngle(Enable := FALSE);
              // move to next step
              seqCtr := 3;
            END_IF;

          // calc step (use looked up angle)
          ELSIF 3 = seqCtr THEN
            // At this point, we have the angle for this pass.
            // This angle is actually the offset angle between the axes.
            // The offset in practice should be negative, meaning the slave lags
            // behind the master by the amount of the offset.
            // Make an entry in the cam table
            // Each pass has an enrty to establish the pass depth,
            // and a second pass to make the cut, which is 1 revolution from the point the
            // depth is established, plus the overcut distance.
            // For a given pass, the first index/position is: ((pass number - 1) * 2) + 1
            // the second index/position is: first index + 1
            // For a given pass, the first master position is: (cutInAngle + pass number) + ((rev + overcut) * (pass number - 1))
            // the second master position is: first position + rev + overcut
            idx := ((passCtr - 1) * 2) + 1; // zero based array index position

            // Establish an offset from previous position
            CamTable.Section[idx].Mode := mcCAMSECTREF_ABSOLUTE;
            CamTable.Section[idx].MasterPoint := (_cutInAngle * passCtr) + ((360.0 + _overCutAngle) * (passCtr - 1));
            CamTable.Section[idx].SlavePoint := CamTable.Section[idx].MasterPoint - passAngle;
            // slave to be at a constant velocity
            CamTable.Section[idx].FirstDerivative := 1.0; // velocity ratio
            CamTable.Section[idx].SecondDerivative := 0.0; // accel ratio
            // next point will be a stright section.
            CamTable.Section[idx].Type := mcCAMSECTLAW_STRAIGHT_LINE;
            CamTable.Section[idx].InflectionPoint := 0.0; // not used for straight line

            // Keep the offset for a revolution + the overcut distance
            CamTable.Section[idx + 1].Mode := mcCAMSECTREF_ABSOLUTE;
            CamTable.Section[idx + 1].MasterPoint := CamTable.Section[idx].MasterPoint + (360.0 + _overCutAngle);
            CamTable.Section[idx + 1].SlavePoint := CamTable.Section[idx + 1].MasterPoint - passAngle;
            // slave to be at a constant velocity
            CamTable.Section[idx + 1].FirstDerivative := 1.0; // velocity ratio
            CamTable.Section[idx + 1].SecondDerivative := 0.0; // accel ratio
            // next point will establish a new offset, so use a polynomial
            CamTable.Section[idx + 1].Type := mcCAMSECTLAW_5TH_ORDER_POLYNOM;
            CamTable.Section[idx + 1].InflectionPoint := 0.0; // not used for polynomial

            // Done with calcs for this pass.
            // Set the sequence counter back to 2 so the next angle can be looked up, and
            // increment the pass count.
            seqCtr := 2;
            passCtr := passCtr + 1;
          END_IF; // seq ctr 2 or 3
        ELSE
          // Done with passes. Ready to move on.
          seqCtr := 4;
        END_IF; // passCtr <= _numPasses
      ELSE // incr cut depth for this pass > 0
        // Special case where finishing pass was entered to be >= final depth.
        // Nothing to do, and this else is here for documentation and as
        // a place holder in case something ends up being needed.
        // The finishing pass is handled next, and will cover this case
        ;
      END_IF // incr cut depth

    ELSIF 4 = seqCtr OR 5 = seqCtr THEN
      // **** Forth step: Lookup the nominal pass angle
      // **** Fifth step: Calculate the nominal pass angle

      // If there is a finishing pass, then create cam entries for it

      // After the for loop, passCount will be 1 more than the number of passes.
      // Perfect for the finishing pass, or the retract entry.
      idx := ((passCtr - 1) * 2) + 1; // zero based array index position
      IF _finishPassDepth > 0.0 THEN
        // There is a finishing pass
        // By definition, the finishing pass gets us to our final depth,
        // so regardless of the earlier passes, the finishing pass is always
        // at the offset to give the final depth.
        // Look up angle for the needed depth
        IF 4 = seqCtr THEN
          // Look up angle for the needed depth
          fbLookupAngle(Enable := TRUE, XVal := _finalDepth);
          IF fbLookupAngle.Done AND NOT fbLookupAngle.Error THEN
            // Lookup was sucessful. Use the looked up value.
            // Force the angle to be positive, as down below the
            // value is subtracted from the master position to force
            // the slave to have a negative offset.
            // Round just for safety so crazy decimal imprecision or rounding does not cause
            // unexpected small differences in cam entries
            passAngle := fctRound3(_I_src := ABS(fbLookupAngle.YVal));
            // done with LU fb
            fbLookupAngle(Enable := FALSE);
            // move to next step
            seqCtr := 5;
          ELSIF fbLookupAngle.Done AND fbLookupAngle.Error THEN
            // Lookup error. Use 0 for the pass angle, and set the error output
            passAngle := 0.0;
            Error := TRUE;
            // done with LU fb
            fbLookupAngle(Enable := FALSE);
            // move to next step
            seqCtr := 5;
          END_IF;

        ELSIF 5 = seqCtr THEN
          // Establish an offset from previous position
          CamTable.Section[idx].Mode := mcCAMSECTREF_ABSOLUTE;
          CamTable.Section[idx].MasterPoint := (_cutInAngle * passCtr) + ((360.0 + _overCutAngle) * (passCtr - 1));
          CamTable.Section[idx].SlavePoint := CamTable.Section[idx].MasterPoint - passAngle;
          // slave to be at a constant velocity
          CamTable.Section[idx].FirstDerivative := 1.0; // velocity ratio
          CamTable.Section[idx].SecondDerivative := 0.0; // accel ratio
          // next point will be a stright section.
          CamTable.Section[idx].Type := mcCAMSECTLAW_STRAIGHT_LINE;
          CamTable.Section[idx].InflectionPoint := 0.0; // not used for straight line

          // Keep the offset for a revolution + the overcut distance
          CamTable.Section[idx + 1].Mode := mcCAMSECTREF_ABSOLUTE;
          CamTable.Section[idx + 1].MasterPoint := CamTable.Section[idx].MasterPoint + (360.0 + _overCutAngle);
          CamTable.Section[idx + 1].SlavePoint := CamTable.Section[idx + 1].MasterPoint - passAngle;
          // slave to be at a constant velocity
          CamTable.Section[idx + 1].FirstDerivative := 1.0; // velocity ratio
          CamTable.Section[idx + 1].SecondDerivative := 0.0; // accel ratio
          // next point will establish a new offset, so use a polynomial
          CamTable.Section[idx + 1].Type := mcCAMSECTLAW_5TH_ORDER_POLYNOM;
          CamTable.Section[idx + 1].InflectionPoint := 0.0; // not used for polynomial

          // increment the pass count so similar it can be used for the last entry
          passCtr := passCtr + 1;
          // calculate a new index for the last entry, which retracts the cutter
          idx := ((passCtr - 1) * 2) + 1; // zero based array index position

          // Done with finishing pass. Ready to move on.
          seqCtr := 6;
        END_IF; // seq ctr 4 or 5
      ELSE
        // _finishPassDepth = <= 0.0 (no finish pass)
        // Ready to move on
        seqCtr := 6;
      END_IF; // _finishPassDepth

    // **** Do the last entry to retract the cutting head.
    // passCount will either be number of passes + 1 in the non-finishing pass case,
    // or will be number of passes + 2 in the finishing pass case. idx and passCount
    // were already adjusted in the finishing pass case.

    ELSIF 6 = seqCtr THEN
      // The last cam entry needs to be of type mcCAMSECTLAW_LAST_POINT
      // Establish a zero offset from previous position
      CamTable.Section[idx].Mode := mcCAMSECTREF_ABSOLUTE;
      CamTable.Section[idx].MasterPoint := (_cutInAngle * passCtr) + ((360.0 + _overCutAngle) * (passCtr - 1));
      CamTable.Section[idx].SlavePoint := CamTable.Section[idx].MasterPoint;
      // slave to be at a constant velocity
      CamTable.Section[idx].FirstDerivative := 1.0; // velocity ratio
      CamTable.Section[idx].SecondDerivative := 0.0; // accel ratio
      // next point will be a stright section.
      CamTable.Section[idx].Type := mcCAMSECTLAW_LAST_POINT;
      CamTable.Section[idx].InflectionPoint := 0.0; // not used for straight line

      // Done with sequence
      Active := FALSE;
      Done := TRUE;
      seqCtr := -1;
    END_IF; // seq ctr
  ELSE
    // Not enabled. Clear OS reset outputs.
    enableOS := FALSE;
    Active := FALSE;
    Done := FALSE;
    Error := FALSE;
  END_IF; // enabled or not

END_FUNCTION_BLOCK

// Given an X, find which of 3 tables to look in
FUNCTION fctGetTableNumberT3
  // Return a 1, 2, or 3 for which table to look in
  // NOTE: X values in each table need to be sorted in ascending order
  // NOTE: It is assumed that x values in table 1 < table 2 < table 3

  // If value is less than or equal the last value in table 1,
  // then the value must represented in or before table 1. Return 1.
  IF xVal <= t1.xVals[t1.numberOfVals - 1] THEN
    fctGetTableNumberT3 := 1;
    RETURN;
  ELSIF xVal >= t3.xVals[0] THEN
    // If value is greater than or equal to the first value in table 3,
    // then the value must be represented in or after table 3. Return 3.
    fctGetTableNumberT3 := 3;
    RETURN;
  ELSE
    // The value must be too big to be represented in table 1,
    // and too small to be represented in table 3.
    // Table 2 is the best choice. Return 2.
    fctGetTableNumberT3 := 2;
    RETURN;
  END_IF;

END_FUNCTION

// Given a table, swap the X and Y values
FUNCTION fctSwapTableT3
  // Make sure number of values does not overrun the array sizes
  length := MIN(SIZEOF(tVals) / SIZEOF(tVals[0]), SIZEOF(table.xVals) / SIZEOF(table.xVals[0]), SIZEOF(table.yVals) / SIZEOF(table.yVals[0]));
  // Y -> temp
  // X -> Y
  // temp -> X
  // nextAddr := brsmemcpy(ADR(Dest),ADR(Src),length);
  nextAddr := brsmemcpy(ADR(tVals), ADR(table.yVals), length);
  nextAddr := brsmemcpy(ADR(table.yVals), ADR(table.xVals), length);
  nextAddr := brsmemcpy(ADR(table.xVals), ADR(tVals), length);
END_FUNCTION
```

Listed in the project but not available here: Logical/Libraries/GAMath/GAMath.typ, Logical/Libraries/GAMath/GAMath.var, Logical/PlcLogic/ProcInputs/ProcInputs.typ, Logical/PlcLogic/CuttingFluidVFD/Types.typ, Logical/PlcLogic/CuttingFluidVFD/Variables.var, Logical/PlcLogic/Annunc/Annunc.typ, Logical/PlcLogic/axSpindle/axSpindle.typ, Logical/PlcLogic/axSpindle/axSpindleSM/AxSMExit.st, Logical/PlcLogic/axSpindle/axSpindleSM/ActionMotionFbs.st, Logical/PlcLogic/axInE/axInE.typ, Logical/PlcLogic/axInE/axInE.var, Logical/PlcLogic/axInE/axInESM/AxSMCyclic.sfc, Logical/PlcLogic/axInE/axInESM/AxSMExit.st, Logical/PlcLogic/axInE/axInESM/ActionChkPermissives.st, Logical/PlcLogic/axInE/axInESM/ActionAxisSpecific.st, Logical/PlcLogic/axZ/axZ.typ, Logical/PlcLogic/axZ/axZ.var, Logical/PlcLogic/axHandwheel/axHw.typ
